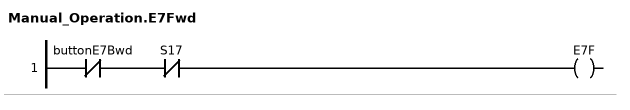
[picture p24: Manual_Operation.E7Fwd (LD)]
_LD_ (* Ladder Diagram *)
NETWORK 1
	[/buttonE7Bwd] - [/S17] --- (E7F)
_END_LD_
(* the same logic as Structured Text *)
(* Network 1 *)
E7F := NOT buttonE7Bwd AND NOT S17;
END_ACTION
ACTION E8Bwd:
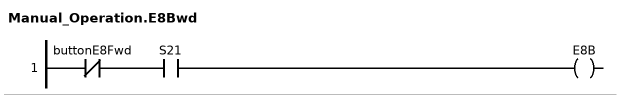
_LD_ (* Ladder Diagram *)
NETWORK 1
	[/buttonE8Fwd] - [S21] --- (E8B)
_END_LD_
(* the same logic as Structured Text *)
(* Network 1 *)
E8B := NOT buttonE8Fwd AND S21;
END_ACTION

(* POU Automatic_Operation, SFC *)
PROGRAM Automatic_Operation
VAR
END_VAR
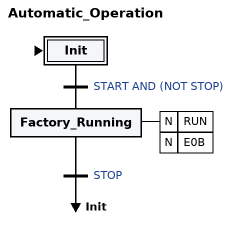
INITIAL_STEP Init:
END_STEP
TRANSITION FROM Init TO Factory_Running := START AND (NOT STOP);
END_TRANSITION
STEP Factory_Running:
	RUN(N);
	E0B(N);
END_STEP
TRANSITION FROM Factory_Running TO Init := STOP;
END_TRANSITION
END_PROGRAM

(* POU Lobby, SFC *)
PROGRAM Lobby
VAR

END_VAR
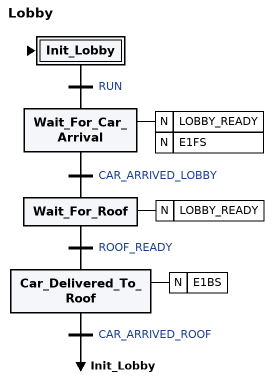
INITIAL_STEP Init_Lobby:
END_STEP
TRANSITION FROM Init_Lobby TO Wait_For_Car_Arrival := RUN;
END_TRANSITION
STEP Wait_For_Car_Arrival:
	LOBBY_READY(N);
	E1FS(N);
END_STEP
TRANSITION FROM Wait_For_Car_Arrival TO Wait_For_Roof := CAR_ARRIVED_LOBBY;
END_TRANSITION
STEP Wait_For_Roof:
	LOBBY_READY(N);
END_STEP
TRANSITION FROM Wait_For_Roof TO Car_Delivered_To_Roof := ROOF_READY;
END_TRANSITION
STEP Car_Delivered_To_Roof:
	E1BS(N);
END_STEP
TRANSITION FROM Car_Delivered_To_Roof TO Init_Lobby := CAR_ARRIVED_ROOF;
END_TRANSITION
END_PROGRAM

(* POU Roof, SFC *)
PROGRAM Roof
VAR
	Roof_Fwd_Go: BOOL;
	Temp_Var_Roof: BOOL;
	LOBBY_DELIVER: BOOL; (*Doesn't do anything rn*)
END_VAR
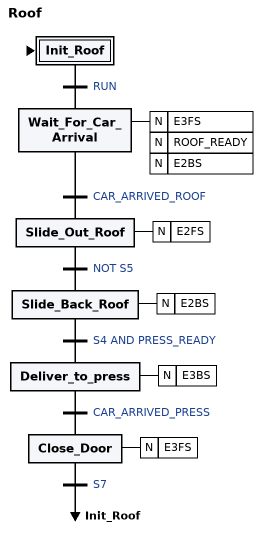
INITIAL_STEP Init_Roof:
END_STEP
TRANSITION FROM Init_Roof TO Wait_For_Car_Arrival := RUN;
END_TRANSITION
STEP Wait_For_Car_Arrival:
	E3FS(N);
	ROOF_READY(N);
	E2BS(N);
END_STEP
TRANSITION FROM Wait_For_Car_Arrival TO Slide_Out_Roof := CAR_ARRIVED_ROOF;
END_TRANSITION
STEP Slide_Out_Roof:
	E2FS(N);
END_STEP
TRANSITION FROM Slide_Out_Roof TO Slide_Back_Roof := NOT S5;
END_TRANSITION
STEP Slide_Back_Roof:
	E2BS(N);
END_STEP
TRANSITION FROM Slide_Back_Roof TO Deliver_to_press := S4 AND PRESS_READY;
END_TRANSITION
STEP Deliver_to_press:
	E3BS(N);
END_STEP
TRANSITION FROM Deliver_to_press TO Close_Door := CAR_ARRIVED_PRESS;
END_TRANSITION
STEP Close_Door:
	E3FS(N);
END_STEP
TRANSITION FROM Close_Door TO Init_Roof := S7;
END_TRANSITION
END_PROGRAM

(* POU Press, SFC *)
PROGRAM Press
VAR
	Temp: BOOL;
END_VAR
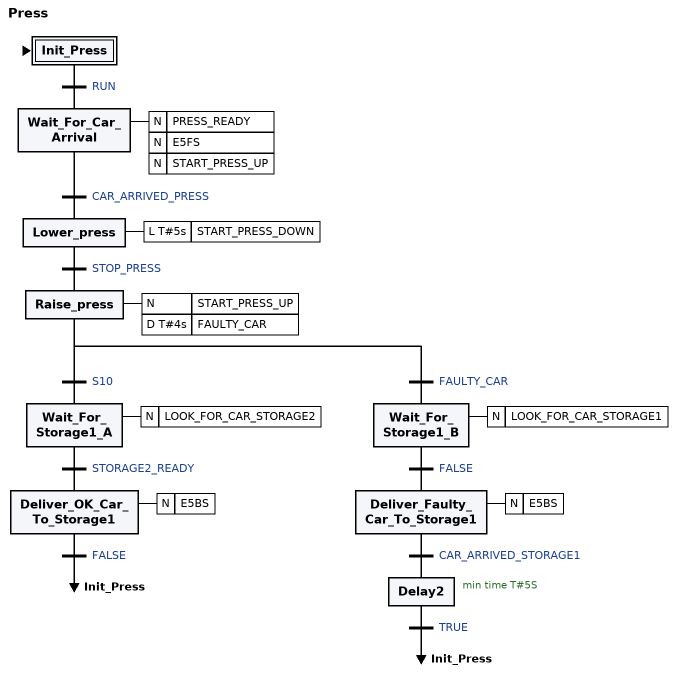
INITIAL_STEP Init_Press:
END_STEP
TRANSITION FROM Init_Press TO Wait_For_Car_Arrival := RUN;
END_TRANSITION
STEP Wait_For_Car_Arrival:
	PRESS_READY(N);
	E5FS(N);
	START_PRESS_UP(N);
END_STEP
TRANSITION FROM Wait_For_Car_Arrival TO Lower_press := CAR_ARRIVED_PRESS;
END_TRANSITION
STEP Lower_press:
	START_PRESS_DOWN(L, T#5s);
END_STEP
TRANSITION FROM Lower_press TO Raise_press := STOP_PRESS;
END_TRANSITION
STEP Raise_press:
	START_PRESS_UP(N);
	FAULTY_CAR(D, T#4s);
END_STEP
TRANSITION FROM Raise_press TO Wait_For_Storage1_A := S10;
END_TRANSITION
TRANSITION FROM Raise_press TO Wait_For_Storage1_B := FAULTY_CAR;
END_TRANSITION
STEP Wait_For_Storage1_A:
	LOOK_FOR_CAR_STORAGE2(N);
END_STEP
TRANSITION FROM Wait_For_Storage1_A TO Deliver_OK_Car_To_Storage1 := STORAGE2_READY;
END_TRANSITION
STEP Wait_For_Storage1_B:
	LOOK_FOR_CAR_STORAGE1(N);
END_STEP
TRANSITION FROM Wait_For_Storage1_B TO Deliver_Faulty_Car_To_Storage1 := FALSE;
END_TRANSITION
STEP Deliver_Faulty_Car_To_Storage1:
	E5BS(N);
END_STEP
TRANSITION FROM Deliver_Faulty_Car_To_Storage1 TO Delay2 := CAR_ARRIVED_STORAGE1;
END_TRANSITION
STEP Delay2: (* min time T#5S *)
END_STEP
TRANSITION FROM Delay2 TO Init_Press := TRUE;
END_TRANSITION
STEP Deliver_OK_Car_To_Storage1:
	E5BS(N);
END_STEP
TRANSITION FROM Deliver_OK_Car_To_Storage1 TO Init_Press := FALSE;
END_TRANSITION
END_PROGRAM

(* POU Storage1, SFC *)
PROGRAM Storage1
VAR
END_VAR
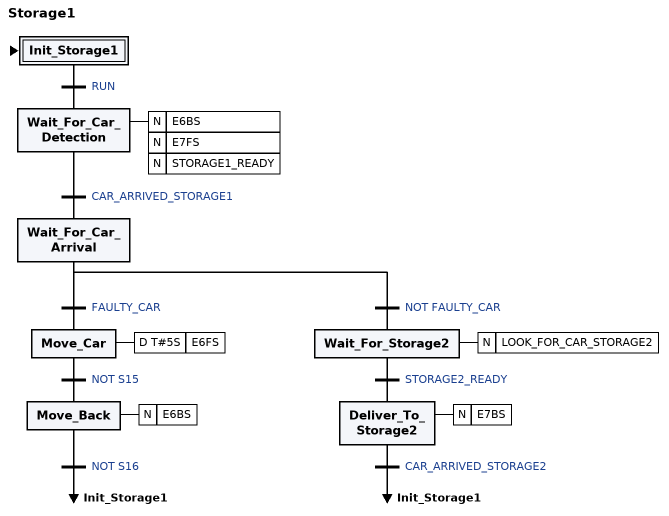
INITIAL_STEP Init_Storage1:
END_STEP
TRANSITION FROM Init_Storage1 TO Wait_For_Car_Detection := RUN;
END_TRANSITION
STEP Wait_For_Car_Detection:
	E6BS(N);
	E7FS(N);
	STORAGE1_READY(N);
END_STEP
TRANSITION FROM Wait_For_Car_Detection TO Wait_For_Car_Arrival := CAR_ARRIVED_STORAGE1;
END_TRANSITION
STEP Wait_For_Car_Arrival:
END_STEP
TRANSITION FROM Wait_For_Car_Arrival TO Move_Car := FAULTY_CAR;
END_TRANSITION
TRANSITION FROM Wait_For_Car_Arrival TO Wait_For_Storage2 := NOT FAULTY_CAR;
END_TRANSITION
STEP Move_Car:
	E6FS(D, T#5S);
END_STEP
TRANSITION FROM Move_Car TO Move_Back := NOT S15;
END_TRANSITION
STEP Move_Back:
	E6BS(N);
END_STEP
TRANSITION FROM Move_Back TO Init_Storage1 := NOT S16;
END_TRANSITION
STEP Wait_For_Storage2:
	LOOK_FOR_CAR_STORAGE2(N);
END_STEP
TRANSITION FROM Wait_For_Storage2 TO Deliver_To_Storage2 := STORAGE2_READY;
END_TRANSITION
STEP Deliver_To_Storage2:
	E7BS(N);
END_STEP
TRANSITION FROM Deliver_To_Storage2 TO Init_Storage1 := CAR_ARRIVED_STORAGE2;
END_TRANSITION
END_PROGRAM

(* POU Storage2, SFC *)
PROGRAM Storage2
VAR
END_VAR
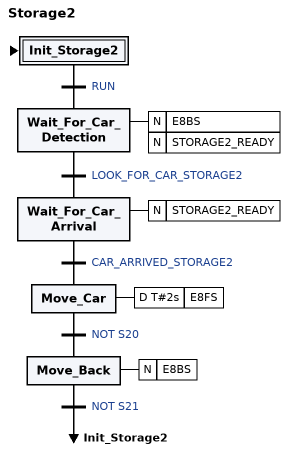
INITIAL_STEP Init_Storage2:
END_STEP
TRANSITION FROM Init_Storage2 TO Wait_For_Car_Detection := RUN;
END_TRANSITION
STEP Wait_For_Car_Detection:
	E8BS(N);
	STORAGE2_READY(N);
END_STEP
TRANSITION FROM Wait_For_Car_Detection TO Wait_For_Car_Arrival := LOOK_FOR_CAR_STORAGE2;
END_TRANSITION
STEP Wait_For_Car_Arrival:
	STORAGE2_READY(N);
END_STEP
TRANSITION FROM Wait_For_Car_Arrival TO Move_Car := CAR_ARRIVED_STORAGE2;
END_TRANSITION
STEP Move_Car:
	E8FS(D, T#2s);
END_STEP
TRANSITION FROM Move_Car TO Move_Back := NOT S20;
END_TRANSITION
STEP Move_Back:
	E8BS(N);
END_STEP
TRANSITION FROM Move_Back TO Init_Storage2 := NOT S21;
END_TRANSITION
END_PROGRAM

(* POU Automatic_Conditional, LD *)
PROGRAM Automatic_Conditional
VAR
	T0: TON;		(*Timer utanför roof*)
	T3: TON;
	T6: TON;
	T9: TON;
	T14: TON; (*Kan behöva tweak:as*)
	T19: TON;
	NOT_START_PRESS_UP: BOOL;
	T_Press: TON;
	TACHO_TRIGGER: R_TRIG;
	Faulty_Car_Time: TON;


END_VAR
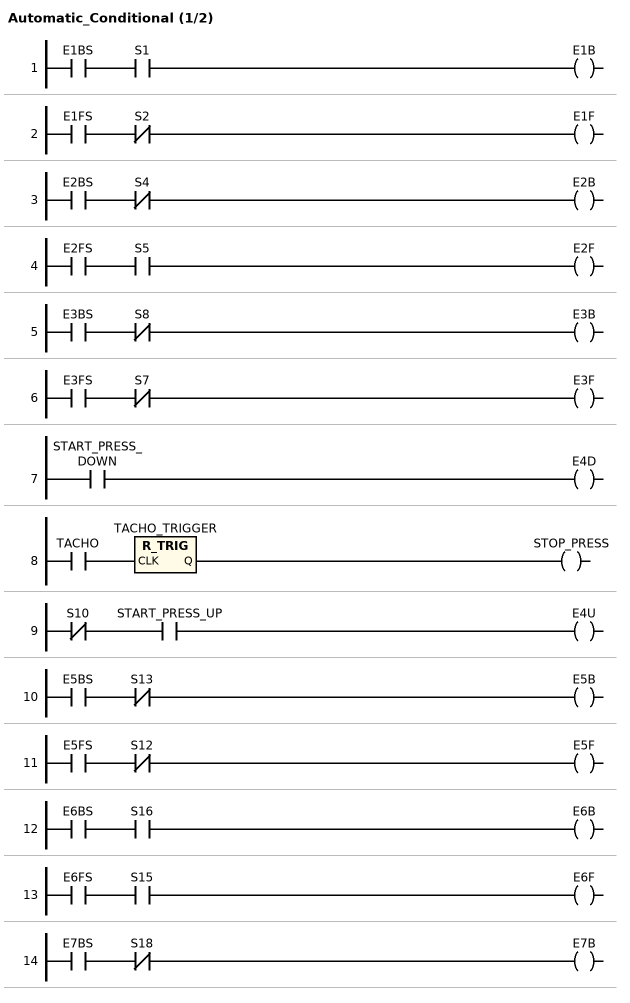
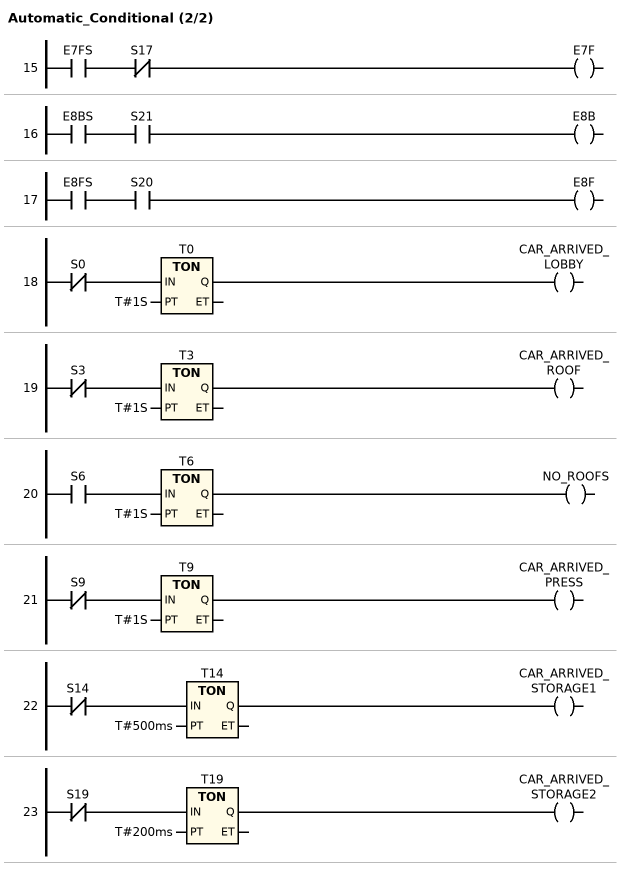
_LD_ (* Ladder Diagram *)
NETWORK 1
	[E1BS] - [S1] --- (E1B)
NETWORK 2
	[E1FS] - [/S2] --- (E1F)
NETWORK 3
	[E2BS] - [/S4] --- (E2B)
NETWORK 4
	[E2FS] - [S5] --- (E2F)
NETWORK 5
	[E3BS] - [/S8] --- (E3B)
NETWORK 6
	[E3FS] - [/S7] --- (E3F)
NETWORK 7
	[START_PRESS_DOWN] --- (E4D)
NETWORK 8
	[TACHO] - TACHO_TRIGGER:R_TRIG(CLK: *) --- (STOP_PRESS)
NETWORK 9
	[/S10] - [START_PRESS_UP] --- (E4U)
NETWORK 10
	[E5BS] - [/S13] --- (E5B)
NETWORK 11
	[E5FS] - [/S12] --- (E5F)
NETWORK 12
	[E6BS] - [S16] --- (E6B)
NETWORK 13
	[E6FS] - [S15] --- (E6F)
NETWORK 14
	[E7BS] - [/S18] --- (E7B)
NETWORK 15
	[E7FS] - [/S17] --- (E7F)
NETWORK 16
	[E8BS] - [S21] --- (E8B)
NETWORK 17
	[E8FS] - [S20] --- (E8F)
NETWORK 18
	[/S0] - T0:TON(IN: *, PT: T#1S) --- (CAR_ARRIVED_LOBBY)
NETWORK 19
	[/S3] - T3:TON(IN: *, PT: T#1S) --- (CAR_ARRIVED_ROOF)
NETWORK 20
	[S6] - T6:TON(IN: *, PT: T#1S) --- (NO_ROOFS)
NETWORK 21
	[/S9] - T9:TON(IN: *, PT: T#1S) --- (CAR_ARRIVED_PRESS)
NETWORK 22
	[/S14] - T14:TON(IN: *, PT: T#500ms) --- (CAR_ARRIVED_STORAGE1)
NETWORK 23
	[/S19] - T19:TON(IN: *, PT: T#200ms) --- (CAR_ARRIVED_STORAGE2)
_END_LD_
(* the same logic as Structured Text *)
(* Network 1 *)
E1B := E1BS AND S1;
(* Network 2 *)
E1F := E1FS AND NOT S2;
(* Network 3 *)
E2B := E2BS AND NOT S4;
(* Network 4 *)
E2F := E2FS AND S5;
(* Network 5 *)
E3B := E3BS AND NOT S8;
(* Network 6 *)
E3F := E3FS AND NOT S7;
(* Network 7 *)
E4D := START_PRESS_DOWN;
(* Network 8 *)
TACHO_TRIGGER(CLK := TACHO);
STOP_PRESS := TACHO_TRIGGER.Q;
(* Network 9 *)
E4U := NOT S10 AND START_PRESS_UP;
(* Network 10 *)
E5B := E5BS AND NOT S13;
(* Network 11 *)
E5F := E5FS AND NOT S12;
(* Network 12 *)
E6B := E6BS AND S16;
(* Network 13 *)
E6F := E6FS AND S15;
(* Network 14 *)
E7B := E7BS AND NOT S18;
(* Network 15 *)
E7F := E7FS AND NOT S17;
(* Network 16 *)
E8B := E8BS AND S21;
(* Network 17 *)
E8F := E8FS AND S20;
(* Network 18 *)
T0(IN := NOT S0, PT := T#1S);
CAR_ARRIVED_LOBBY := T0.Q;
(* Network 19 *)
T3(IN := NOT S3, PT := T#1S);
CAR_ARRIVED_ROOF := T3.Q;
(* Network 20 *)
T6(IN := S6, PT := T#1S);
NO_ROOFS := T6.Q;
(* Network 21 *)
T9(IN := NOT S9, PT := T#1S);
CAR_ARRIVED_PRESS := T9.Q;
(* Network 22 *)
T14(IN := NOT S14, PT := T#500ms);
CAR_ARRIVED_STORAGE1 := T14.Q;
(* Network 23 *)
T19(IN := NOT S19, PT := T#200ms);
CAR_ARRIVED_STORAGE2 := T19.Q;
END_PROGRAM
